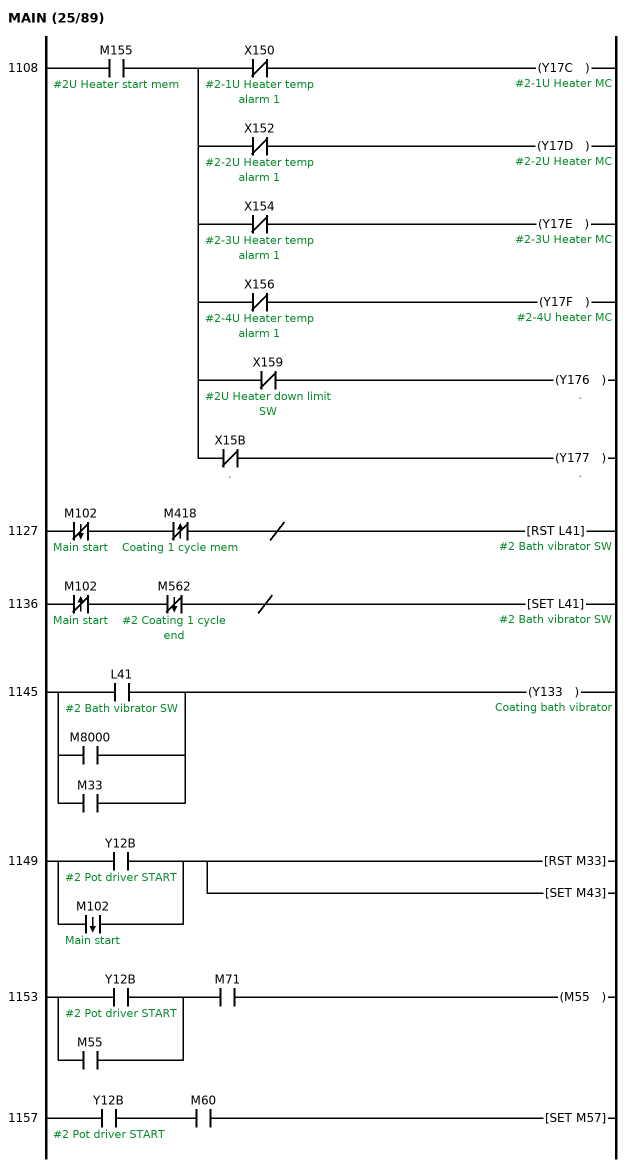
[picture p24: ladder of MAIN, rungs at steps 1108 to 1157]
1108  LD      M155  ; #2U Heater start mem
      MPS
      ANI     X150  ; #2-1U Heater temp alarm 1
      OUT     Y17C  ; #2-1U Heater MC
      MRD
      ANI     X152  ; #2-2U Heater temp alarm 1
      OUT     Y17D  ; #2-2U Heater MC
      MRD
      ANI     X154  ; #2-3U Heater temp alarm 1
      OUT     Y17E  ; #2-3U Heater MC
      MRD
      ANI     X156  ; #2-4U Heater temp alarm 1
      OUT     Y17F  ; #2-4U heater MC
      MRD
      ANI     X159  ; #2U Heater down limit SW
      OUT     Y176  ; .
      MPP
      ANI     X15B  ; .
      OUT     Y177  ; .
1127  LDFI    M102  ; Main start
      ANDPI   M418  ; Coating 1 cycle mem
      INV
      RST     L41  ; #2 Bath vibrator SW
1136  LDPI    M102  ; Main start
      ANDFI   M562  ; #2 Coating 1 cycle end
      INV
      SET     L41  ; #2 Bath vibrator SW
1145  LD      L41  ; #2 Bath vibrator SW
      OR      M8000
      OR      M33
      OUT     Y133  ; Coating bath vibrator
1149  LD      Y12B  ; #2 Pot driver START
      ORF     M102  ; Main start
      RST     M33
      SET     M43
1153  LD      Y12B  ; #2 Pot driver START
      OR      M55
      AND     M71
      OUT     M55
1157  LD      Y12B  ; #2 Pot driver START
      AND     M60
      SET     M57
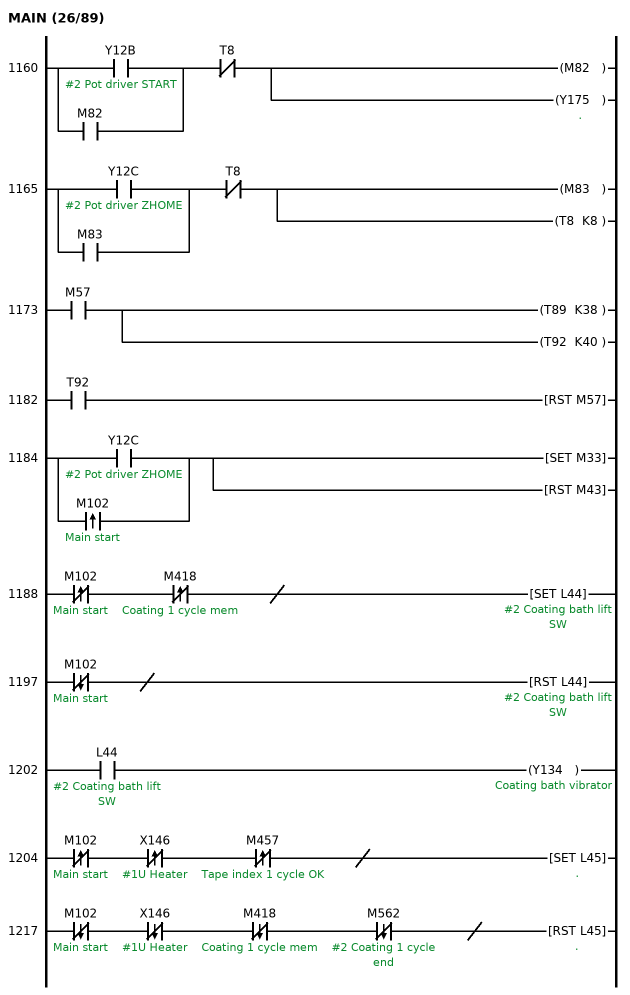
1160  LD      Y12B  ; #2 Pot driver START
      OR      M82
      ANI     T8
      OUT     M82
      OUT     Y175  ; .
1165  LD      Y12C  ; #2 Pot driver ZHOME
      OR      M83
      ANI     T8
      OUT     M83
      OUT     T8 K8
1173  LD      M57
      OUT     T89 K38
      OUT     T92 K40
1182  LD      T92
      RST     M57
1184  LD      Y12C  ; #2 Pot driver ZHOME
      ORP     M102  ; Main start
      SET     M33
      RST     M43
1188  LDPI    M102  ; Main start
      ANDPI   M418  ; Coating 1 cycle mem
      INV
      SET     L44  ; #2 Coating bath lift SW
1197  LDFI    M102  ; Main start
      INV
      RST     L44  ; #2 Coating bath lift SW
1202  LD      L44  ; #2 Coating bath lift SW
      OUT     Y134  ; Coating bath vibrator
1204  LDPI    M102  ; Main start
      ANDPI   X146  ; #1U Heater
      ANDPI   M457  ; Tape index 1 cycle OK
      INV
      SET     L45  ; .
1217  LDFI    M102  ; Main start
      ANDFI   X146  ; #1U Heater
      ANDFI   M418  ; Coating 1 cycle mem
      ANDFI   M562  ; #2 Coating 1 cycle end
      INV
      RST     L45  ; .
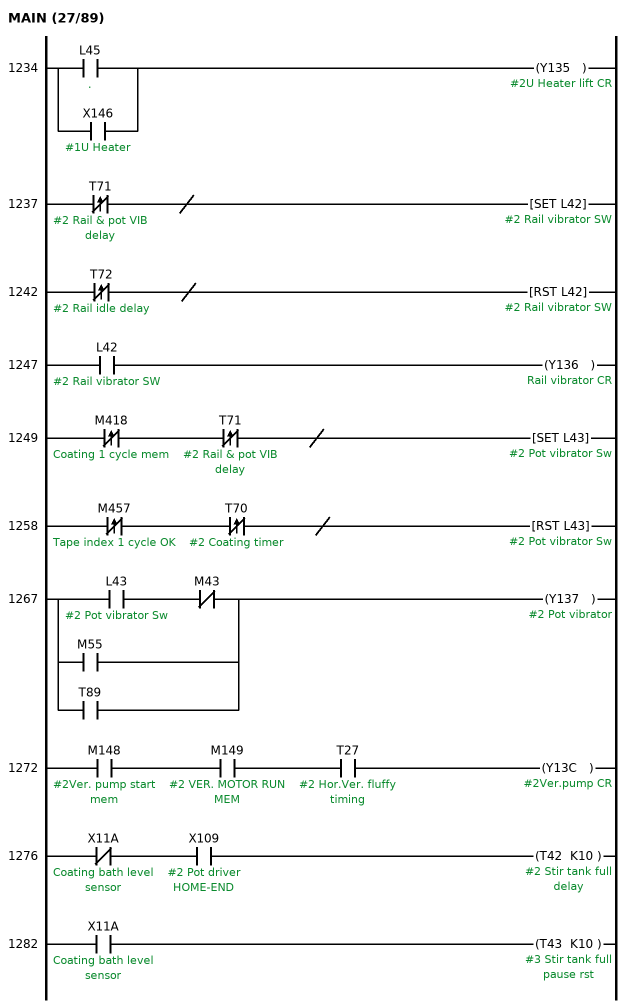
1234  LD      L45  ; .
      OR      X146  ; #1U Heater
      OUT     Y135  ; #2U Heater lift CR
1237  LDPI    T71  ; #2 Rail & pot VIB delay
      INV
      SET     L42  ; #2 Rail vibrator SW
1242  LDPI    T72  ; #2 Rail idle delay
      INV
      RST     L42  ; #2 Rail vibrator SW
1247  LD      L42  ; #2 Rail vibrator SW
      OUT     Y136  ; Rail vibrator CR
1249  LDPI    M418  ; Coating 1 cycle mem
      ANDPI   T71  ; #2 Rail & pot VIB delay
      INV
      SET     L43  ; #2 Pot vibrator Sw
1258  LDPI    M457  ; Tape index 1 cycle OK
      ANDPI   T70  ; #2 Coating timer
      INV
      RST     L43  ; #2 Pot vibrator Sw
1267  LD      L43  ; #2 Pot vibrator Sw
      ANI     M43
      OR      M55
      OR      T89
      OUT     Y137  ; #2 Pot vibrator
1272  LD      M148  ; #2Ver. pump start mem
      AND     M149  ; #2 VER. MOTOR RUN MEM
      AND     T27  ; #2 Hor.Ver. fluffy timing
      OUT     Y13C  ; #2Ver.pump CR
1276  LDI     X11A  ; Coating bath level sensor
      AND     X109  ; #2 Pot driver HOME-END
      OUT     T42 K10  ; #2 Stir tank full delay
1282  LD      X11A  ; Coating bath level sensor
      OUT     T43 K10  ; #3 Stir tank full pause rst
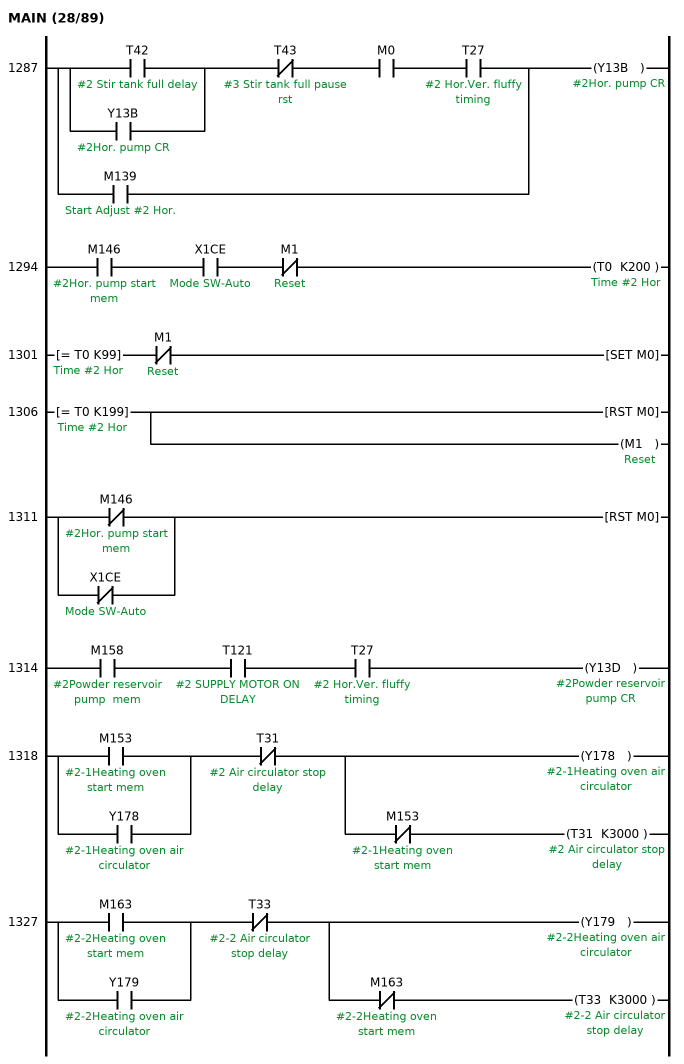
1287  LD      T42  ; #2 Stir tank full delay
      OR      Y13B  ; #2Hor. pump CR
      ANI     T43  ; #3 Stir tank full pause rst
      AND     M0
      AND     T27  ; #2 Hor.Ver. fluffy timing
      OR      M139  ; Start Adjust #2 Hor.
      OUT     Y13B  ; #2Hor. pump CR
1294  LD      M146  ; #2Hor. pump start mem
      AND     X1CE  ; Mode SW-Auto
      ANI     M1  ; Reset
      OUT     T0 K200  ; Time #2 Hor
1301  LD=     T0 K99  ; Time #2 Hor
      ANI     M1  ; Reset
      SET     M0
1306  LD=     T0 K199  ; Time #2 Hor
      RST     M0
      OUT     M1  ; Reset
1311  LDI     M146  ; #2Hor. pump start mem
      ORI     X1CE  ; Mode SW-Auto
      RST     M0
1314  LD      M158  ; #2Powder reservoir pump  mem
      AND     T121  ; #2 SUPPLY MOTOR ON DELAY
      AND     T27  ; #2 Hor.Ver. fluffy timing
      OUT     Y13D  ; #2Powder reservoir pump CR
1318  LD      M153  ; #2-1Heating oven start mem
      OR      Y178  ; #2-1Heating oven air circulator
      ANI     T31  ; #2 Air circulator stop delay
      OUT     Y178  ; #2-1Heating oven air circulator
      ANI     M153  ; #2-1Heating oven start mem
      OUT     T31 K3000  ; #2 Air circulator stop delay
1327  LD      M163  ; #2-2Heating oven start mem
      OR      Y179  ; #2-2Heating oven air circulator
      ANI     T33  ; #2-2 Air circulator stop delay
      OUT     Y179  ; #2-2Heating oven air circulator
      ANI     M163  ; #2-2Heating oven start mem
      OUT     T33 K3000  ; #2-2 Air circulator stop delay
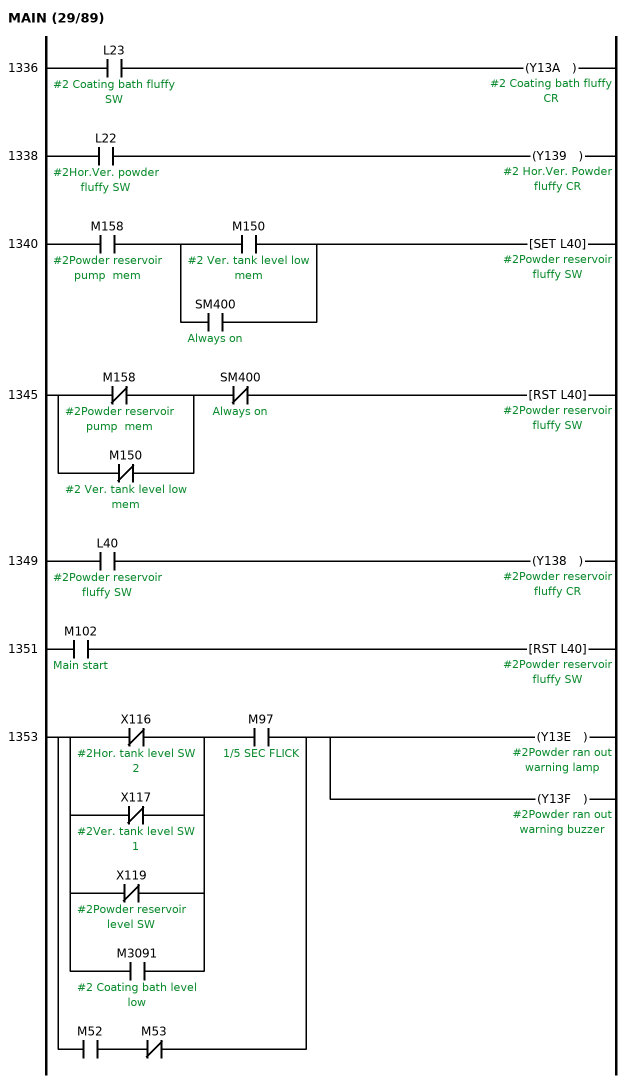
1336  LD      L23  ; #2 Coating bath fluffy SW
      OUT     Y13A  ; #2 Coating bath fluffy CR
1338  LD      L22  ; #2Hor.Ver. powder fluffy SW
      OUT     Y139  ; #2 Hor.Ver. Powder fluffy CR
1340  LD      M158  ; #2Powder reservoir pump  mem
      LD      M150  ; #2 Ver. tank level low mem
      OR      SM400  ; Always on
      ANB
      SET     L40  ; #2Powder reservoir fluffy SW
1345  LDI     M158  ; #2Powder reservoir pump  mem
      ORI     M150  ; #2 Ver. tank level low mem
      ANI     SM400  ; Always on
      RST     L40  ; #2Powder reservoir fluffy SW
1349  LD      L40  ; #2Powder reservoir fluffy SW
      OUT     Y138  ; #2Powder reservoir fluffy CR
1351  LD      M102  ; Main start
      RST     L40  ; #2Powder reservoir fluffy SW
1353  LDI     X116  ; #2Hor. tank level SW 2
      ORI     X117  ; #2Ver. tank level SW 1
      ORI     X119  ; #2Powder reservoir level SW
      OR      M3091  ; #2 Coating bath level low
      AND     M97  ; 1/5 SEC FLICK
      LD      M52
      ANI     M53
      ORB
      OUT     Y13E  ; #2Powder ran out warning lamp
      OUT     Y13F  ; #2Powder ran out warning buzzer
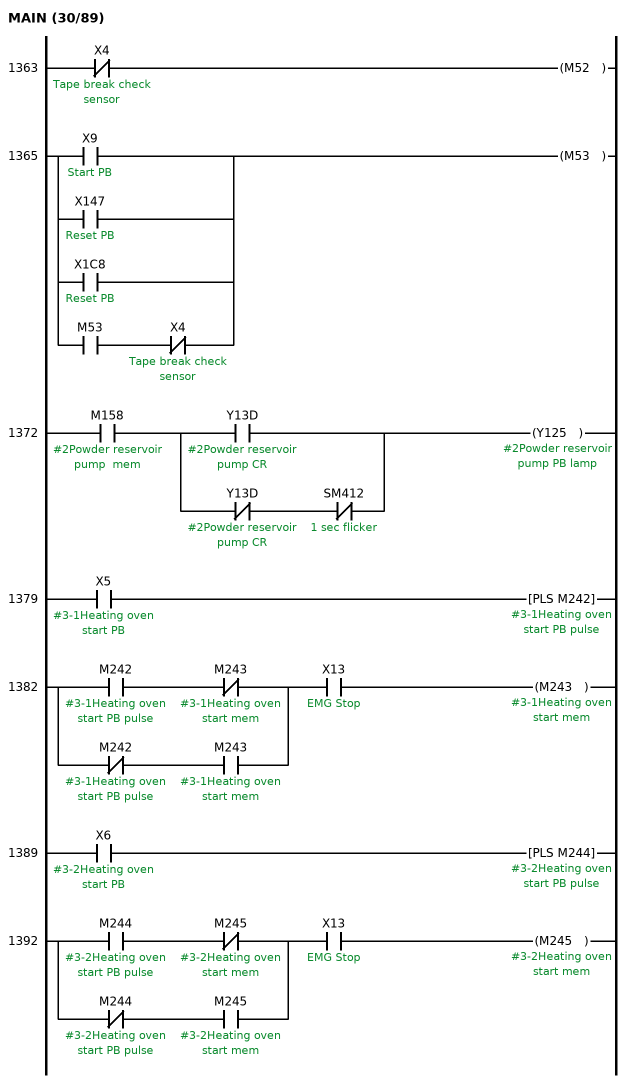
1363  LDI     X4  ; Tape break check sensor
      OUT     M52
1365  LD      X9  ; Start PB
      OR      X147  ; Reset PB
      OR      X1C8  ; Reset PB
      LD      M53
      ANI     X4  ; Tape break check sensor
      ORB
      OUT     M53
1372  LD      M158  ; #2Powder reservoir pump  mem
      LD      Y13D  ; #2Powder reservoir pump CR
      LDI     Y13D  ; #2Powder reservoir pump CR
      ANI     SM412  ; 1 sec flicker
      ORB
      ANB
      OUT     Y125  ; #2Powder reservoir pump PB lamp
1379  LD      X5  ; #3-1Heating oven start PB
      PLS     M242  ; #3-1Heating oven start PB pulse
1382  LD      M242  ; #3-1Heating oven start PB pulse
      ANI     M243  ; #3-1Heating oven start mem
      LDI     M242  ; #3-1Heating oven start PB pulse
      AND     M243  ; #3-1Heating oven start mem
      ORB
      AND     X13  ; EMG Stop
      OUT     M243  ; #3-1Heating oven start mem
1389  LD      X6  ; #3-2Heating oven start PB
      PLS     M244  ; #3-2Heating oven start PB pulse
1392  LD      M244  ; #3-2Heating oven start PB pulse
      ANI     M245  ; #3-2Heating oven start mem
      LDI     M244  ; #3-2Heating oven start PB pulse
      AND     M245  ; #3-2Heating oven start mem
      ORB
      AND     X13  ; EMG Stop
      OUT     M245  ; #3-2Heating oven start mem
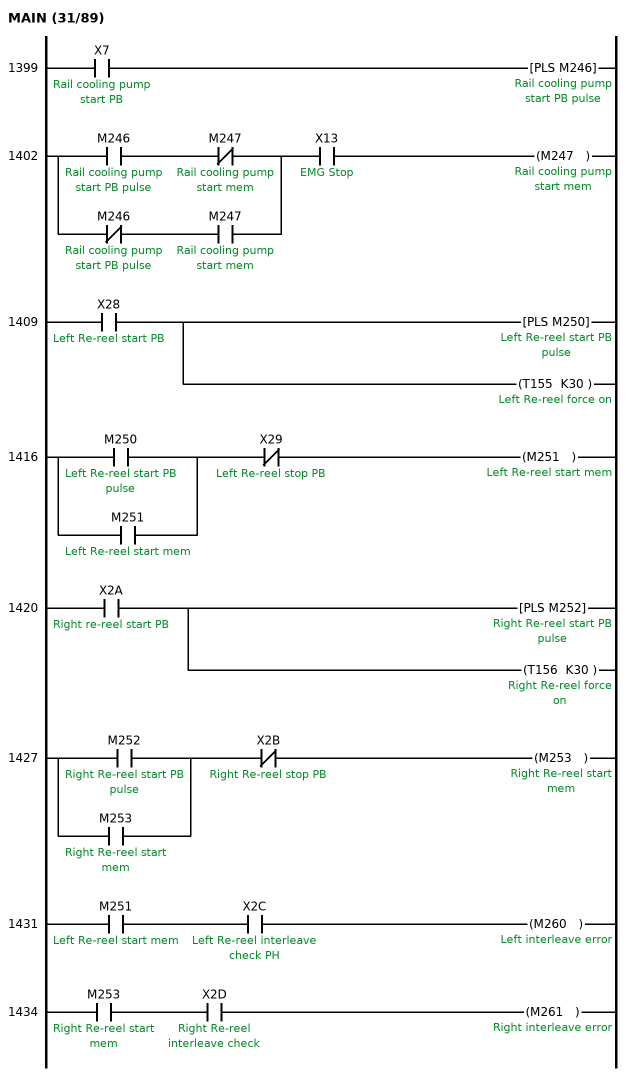
1399  LD      X7  ; Rail cooling pump start PB
      PLS     M246  ; Rail cooling pump start PB pulse
1402  LD      M246  ; Rail cooling pump start PB pulse
      ANI     M247  ; Rail cooling pump start mem
      LDI     M246  ; Rail cooling pump start PB pulse
      AND     M247  ; Rail cooling pump start mem
      ORB
      AND     X13  ; EMG Stop
      OUT     M247  ; Rail cooling pump start mem
1409  LD      X28  ; Left Re-reel start PB
      PLS     M250  ; Left Re-reel start PB pulse
      OUT     T155 K30  ; Left Re-reel force on
1416  LD      M250  ; Left Re-reel start PB pulse
      OR      M251  ; Left Re-reel start mem
      ANI     X29  ; Left Re-reel stop PB
      OUT     M251  ; Left Re-reel start mem
1420  LD      X2A  ; Right re-reel start PB
      PLS     M252  ; Right Re-reel start PB pulse
      OUT     T156 K30  ; Right Re-reel force on
1427  LD      M252  ; Right Re-reel start PB pulse
      OR      M253  ; Right Re-reel start mem
      ANI     X2B  ; Right Re-reel stop PB
      OUT     M253  ; Right Re-reel start mem
1431  LD      M251  ; Left Re-reel start mem
      AND     X2C  ; Left Re-reel interleave check PH
      OUT     M260  ; Left interleave error
1434  LD      M253  ; Right Re-reel start mem
      AND     X2D  ; Right Re-reel interleave check
      OUT     M261  ; Right interleave error
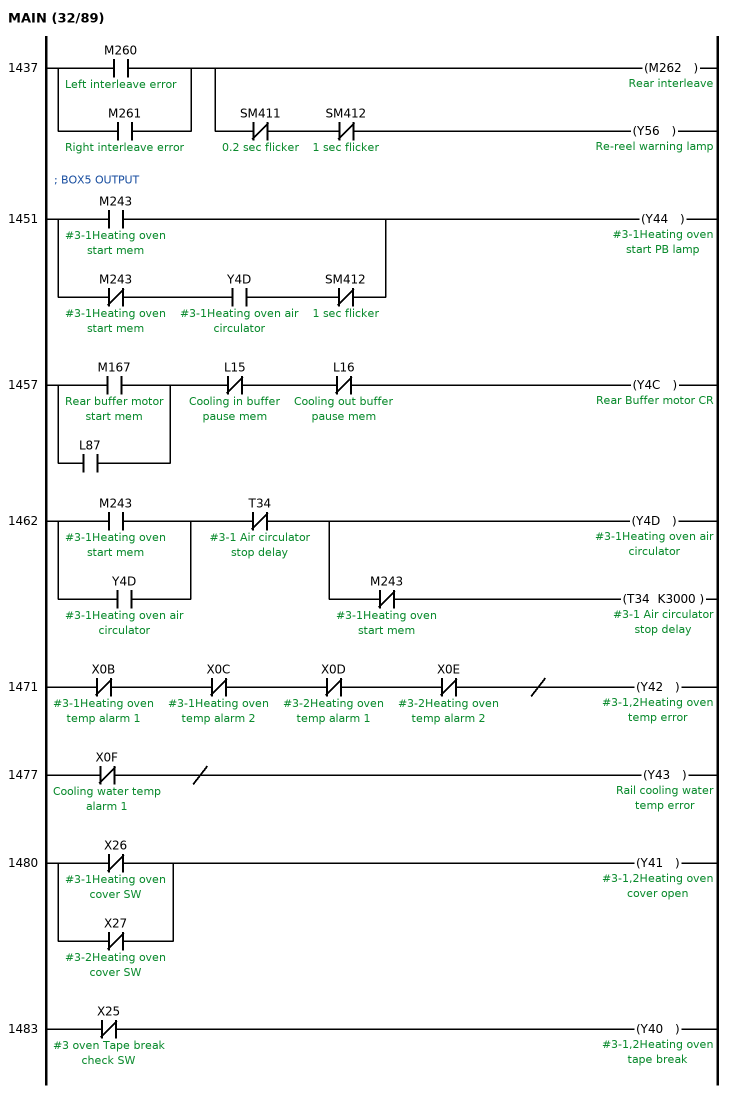
1437  LD      M260  ; Left interleave error
      OR      M261  ; Right interleave error
      OUT     M262  ; Rear interleave
      ANI     SM411  ; 0.2 sec flicker
      ANI     SM412  ; 1 sec flicker
      OUT     Y56  ; Re-reel warning lamp
; BOX5 OUTPUT
1451  LD      M243  ; #3-1Heating oven start mem
      LDI     M243  ; #3-1Heating oven start mem
      AND     Y4D  ; #3-1Heating oven air circulator
      ANI     SM412  ; 1 sec flicker
      ORB
      OUT     Y44  ; #3-1Heating oven start PB lamp
1457  LD      M167  ; Rear buffer motor start mem
      OR      L87
      ANI     L15  ; Cooling in buffer pause mem
      ANI     L16  ; Cooling out buffer pause mem
      OUT     Y4C  ; Rear Buffer motor CR
1462  LD      M243  ; #3-1Heating oven start mem
      OR      Y4D  ; #3-1Heating oven air circulator
      ANI     T34  ; #3-1 Air circulator stop delay
      OUT     Y4D  ; #3-1Heating oven air circulator
      ANI     M243  ; #3-1Heating oven start mem
      OUT     T34 K3000  ; #3-1 Air circulator stop delay
1471  LDI     X0B  ; #3-1Heating oven temp alarm 1
      ANI     X0C  ; #3-1Heating oven temp alarm 2
      ANI     X0D  ; #3-2Heating oven temp alarm 1
      ANI     X0E  ; #3-2Heating oven temp alarm 2
      INV
      OUT     Y42  ; #3-1,2Heating oven temp error
1477  LDI     X0F  ; Cooling water temp alarm 1
      INV
      OUT     Y43  ; Rail cooling water temp error
1480  LDI     X26  ; #3-1Heating oven cover SW
      ORI     X27  ; #3-2Heating oven cover SW
      OUT     Y41  ; #3-1,2Heating oven cover open
1483  LDI     X25  ; #3 oven Tape break check SW
      OUT     Y40  ; #3-1,2Heating oven tape break
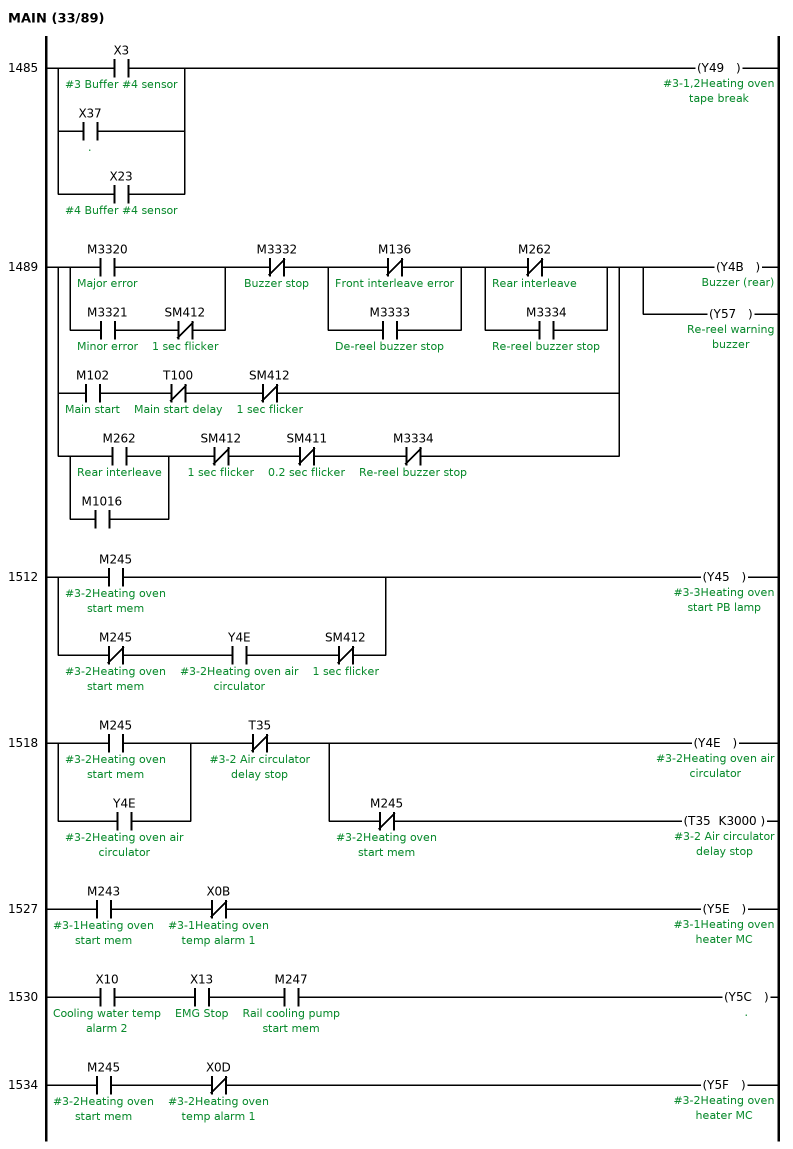
1485  LD      X3  ; #3 Buffer #4 sensor
      OR      X37  ; .
      OR      X23  ; #4 Buffer #4 sensor
      OUT     Y49  ; #3-1,2Heating oven tape break
1489  LD      M3320  ; Major error
      LD      M3321  ; Minor error
      ANI     SM412  ; 1 sec flicker
      ORB
      ANI     M3332  ; Buzzer stop
      LDI     M136  ; Front interleave error
      OR      M3333  ; De-reel buzzer stop
      ANB
      LDI     M262  ; Rear interleave
      OR      M3334  ; Re-reel buzzer stop
      ANB
      LD      M102  ; Main start
      ANI     T100  ; Main start delay
      ANI     SM412  ; 1 sec flicker
      ORB
      LD      M262  ; Rear interleave
      OR      M1016
      ANI     SM412  ; 1 sec flicker
      ANI     SM411  ; 0.2 sec flicker
      ANI     M3334  ; Re-reel buzzer stop
      ORB
      OUT     Y4B  ; Buzzer (rear)
      OUT     Y57  ; Re-reel warning buzzer
1512  LD      M245  ; #3-2Heating oven start mem
      LDI     M245  ; #3-2Heating oven start mem
      AND     Y4E  ; #3-2Heating oven air circulator
      ANI     SM412  ; 1 sec flicker
      ORB
      OUT     Y45  ; #3-3Heating oven start PB lamp
1518  LD      M245  ; #3-2Heating oven start mem
      OR      Y4E  ; #3-2Heating oven air circulator
      ANI     T35  ; #3-2 Air circulator delay stop
      OUT     Y4E  ; #3-2Heating oven air circulator
      ANI     M245  ; #3-2Heating oven start mem
      OUT     T35 K3000  ; #3-2 Air circulator delay stop
1527  LD      M243  ; #3-1Heating oven start mem
      ANI     X0B  ; #3-1Heating oven temp alarm 1
      OUT     Y5E  ; #3-1Heating oven heater MC
1530  LD      X10  ; Cooling water temp alarm 2
      AND     X13  ; EMG Stop
      AND     M247  ; Rail cooling pump start mem
      OUT     Y5C  ; .
1534  LD      M245  ; #3-2Heating oven start mem
      ANI     X0D  ; #3-2Heating oven temp alarm 1
      OUT     Y5F  ; #3-2Heating oven heater MC
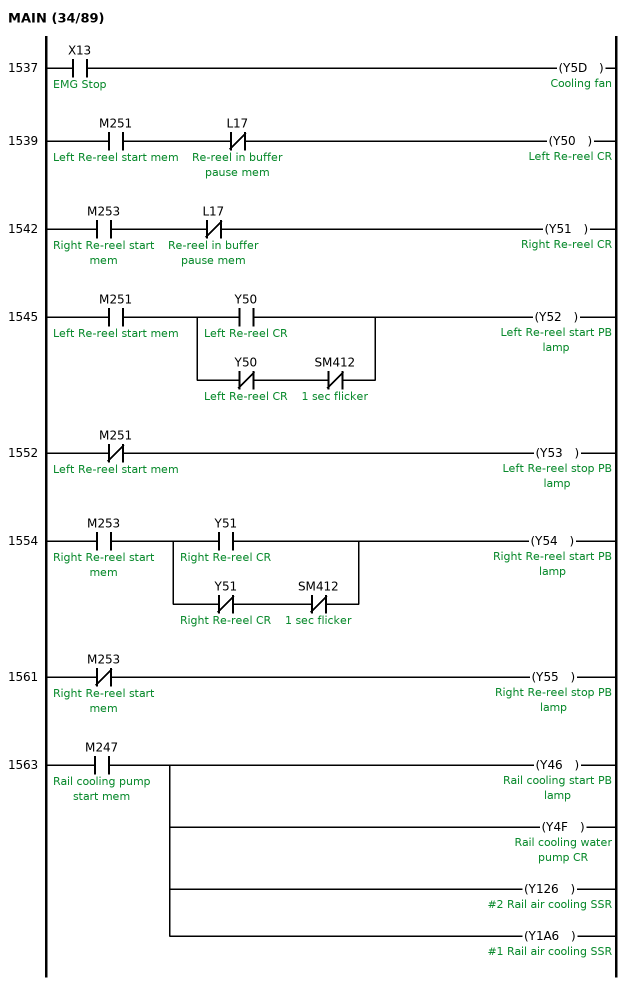
1537  LD      X13  ; EMG Stop
      OUT     Y5D  ; Cooling fan
1539  LD      M251  ; Left Re-reel start mem
      ANI     L17  ; Re-reel in buffer pause mem
      OUT     Y50  ; Left Re-reel CR
1542  LD      M253  ; Right Re-reel start mem
      ANI     L17  ; Re-reel in buffer pause mem
      OUT     Y51  ; Right Re-reel CR
1545  LD      M251  ; Left Re-reel start mem
      LD      Y50  ; Left Re-reel CR
      LDI     Y50  ; Left Re-reel CR
      ANI     SM412  ; 1 sec flicker
      ORB
      ANB
      OUT     Y52  ; Left Re-reel start PB lamp
1552  LDI     M251  ; Left Re-reel start mem
      OUT     Y53  ; Left Re-reel stop PB lamp
1554  LD      M253  ; Right Re-reel start mem
      LD      Y51  ; Right Re-reel CR
      LDI     Y51  ; Right Re-reel CR
      ANI     SM412  ; 1 sec flicker
      ORB
      ANB
      OUT     Y54  ; Right Re-reel start PB lamp
1561  LDI     M253  ; Right Re-reel start mem
      OUT     Y55  ; Right Re-reel stop PB lamp
1563  LD      M247  ; Rail cooling pump start mem
      OUT     Y46  ; Rail cooling start PB lamp
      OUT     Y4F  ; Rail cooling water pump CR
      OUT     Y126  ; #2 Rail air cooling SSR
      OUT     Y1A6  ; #1 Rail air cooling SSR
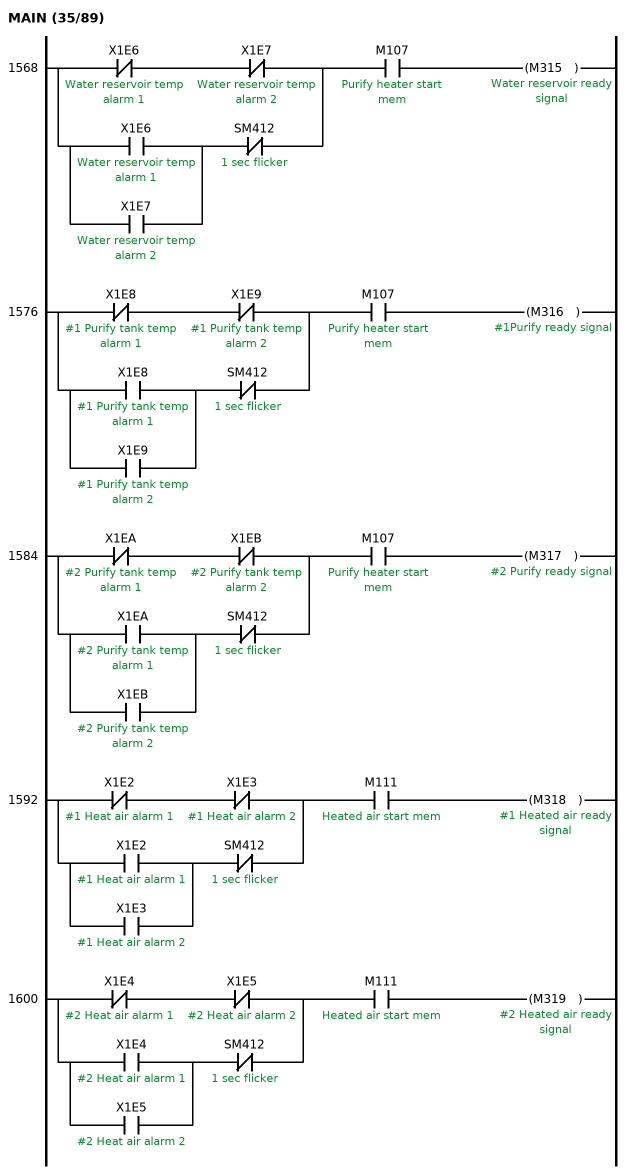
1568  LDI     X1E6  ; Water reservoir temp alarm 1
      ANI     X1E7  ; Water reservoir temp alarm 2
      LD      X1E6  ; Water reservoir temp alarm 1
      OR      X1E7  ; Water reservoir temp alarm 2
      ANI     SM412  ; 1 sec flicker
      ORB
      AND     M107  ; Purify heater start mem
      OUT     M315  ; Water reservoir ready signal
1576  LDI     X1E8  ; #1 Purify tank temp alarm 1
      ANI     X1E9  ; #1 Purify tank temp alarm 2
      LD      X1E8  ; #1 Purify tank temp alarm 1
      OR      X1E9  ; #1 Purify tank temp alarm 2
      ANI     SM412  ; 1 sec flicker
      ORB
      AND     M107  ; Purify heater start mem
      OUT     M316  ; #1Purify ready signal
1584  LDI     X1EA  ; #2 Purify tank temp alarm 1
      ANI     X1EB  ; #2 Purify tank temp alarm 2
      LD      X1EA  ; #2 Purify tank temp alarm 1
      OR      X1EB  ; #2 Purify tank temp alarm 2
      ANI     SM412  ; 1 sec flicker
      ORB
      AND     M107  ; Purify heater start mem
      OUT     M317  ; #2 Purify ready signal
1592  LDI     X1E2  ; #1 Heat air alarm 1
      ANI     X1E3  ; #1 Heat air alarm 2
      LD      X1E2  ; #1 Heat air alarm 1
      OR      X1E3  ; #1 Heat air alarm 2
      ANI     SM412  ; 1 sec flicker
      ORB
      AND     M111  ; Heated air start mem
      OUT     M318  ; #1 Heated air ready signal
1600  LDI     X1E4  ; #2 Heat air alarm 1
      ANI     X1E5  ; #2 Heat air alarm 2
      LD      X1E4  ; #2 Heat air alarm 1
      OR      X1E5  ; #2 Heat air alarm 2
      ANI     SM412  ; 1 sec flicker
      ORB
      AND     M111  ; Heated air start mem
      OUT     M319  ; #2 Heated air ready signal
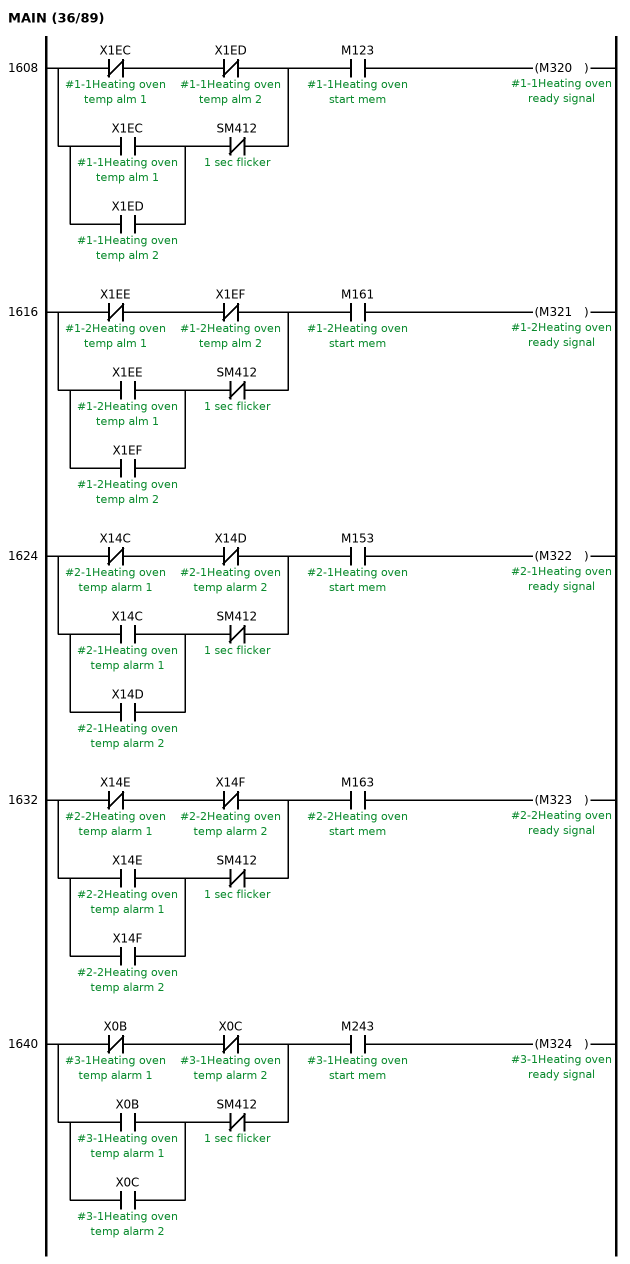
1608  LDI     X1EC  ; #1-1Heating oven temp alm 1
      ANI     X1ED  ; #1-1Heating oven temp alm 2
      LD      X1EC  ; #1-1Heating oven temp alm 1
      OR      X1ED  ; #1-1Heating oven temp alm 2
      ANI     SM412  ; 1 sec flicker
      ORB
      AND     M123  ; #1-1Heating oven start mem
      OUT     M320  ; #1-1Heating oven ready signal
1616  LDI     X1EE  ; #1-2Heating oven temp alm 1
      ANI     X1EF  ; #1-2Heating oven temp alm 2
      LD      X1EE  ; #1-2Heating oven temp alm 1
      OR      X1EF  ; #1-2Heating oven temp alm 2
      ANI     SM412  ; 1 sec flicker
      ORB
      AND     M161  ; #1-2Heating oven start mem
      OUT     M321  ; #1-2Heating oven ready signal
1624  LDI     X14C  ; #2-1Heating oven temp alarm 1
      ANI     X14D  ; #2-1Heating oven temp alarm 2
      LD      X14C  ; #2-1Heating oven temp alarm 1
      OR      X14D  ; #2-1Heating oven temp alarm 2
      ANI     SM412  ; 1 sec flicker
      ORB
      AND     M153  ; #2-1Heating oven start mem
      OUT     M322  ; #2-1Heating oven ready signal
1632  LDI     X14E  ; #2-2Heating oven temp alarm 1
      ANI     X14F  ; #2-2Heating oven temp alarm 2
      LD      X14E  ; #2-2Heating oven temp alarm 1
      OR      X14F  ; #2-2Heating oven temp alarm 2
      ANI     SM412  ; 1 sec flicker
      ORB
      AND     M163  ; #2-2Heating oven start mem
      OUT     M323  ; #2-2Heating oven ready signal
1640  LDI     X0B  ; #3-1Heating oven temp alarm 1
      ANI     X0C  ; #3-1Heating oven temp alarm 2
      LD      X0B  ; #3-1Heating oven temp alarm 1
      OR      X0C  ; #3-1Heating oven temp alarm 2
      ANI     SM412  ; 1 sec flicker
      ORB
      AND     M243  ; #3-1Heating oven start mem
      OUT     M324  ; #3-1Heating oven ready signal
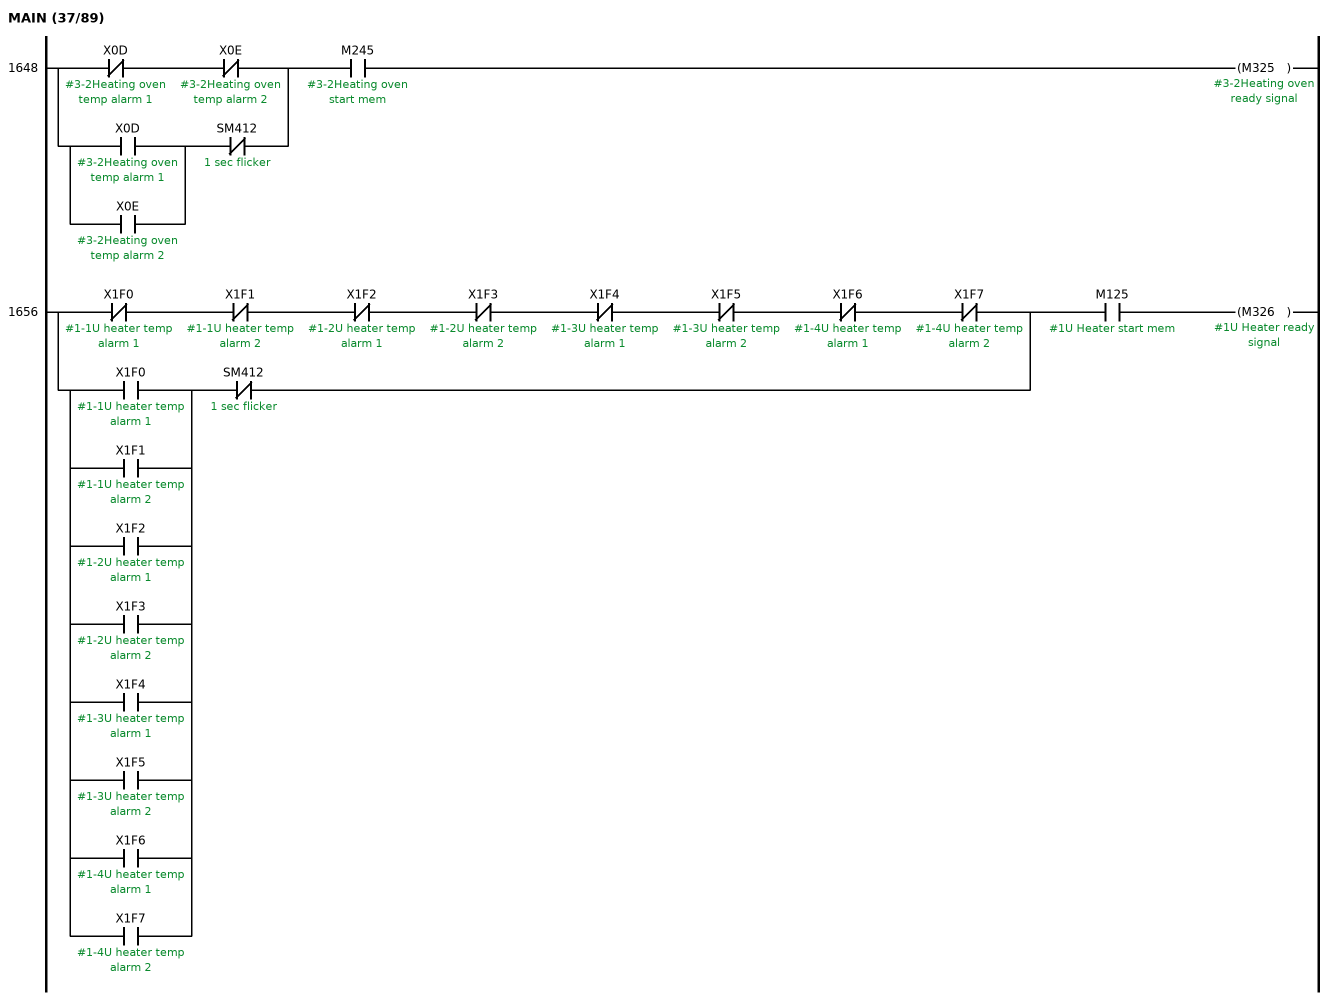
1648  LDI     X0D  ; #3-2Heating oven temp alarm 1
      ANI     X0E  ; #3-2Heating oven temp alarm 2
      LD      X0D  ; #3-2Heating oven temp alarm 1
      OR      X0E  ; #3-2Heating oven temp alarm 2
      ANI     SM412  ; 1 sec flicker
      ORB
      AND     M245  ; #3-2Heating oven start mem
      OUT     M325  ; #3-2Heating oven ready signal
1656  LDI     X1F0  ; #1-1U heater temp alarm 1
      ANI     X1F1  ; #1-1U heater temp alarm 2
      ANI     X1F2  ; #1-2U heater temp alarm 1
      ANI     X1F3  ; #1-2U heater temp alarm 2
      ANI     X1F4  ; #1-3U heater temp alarm 1
      ANI     X1F5  ; #1-3U heater temp alarm 2
      ANI     X1F6  ; #1-4U heater temp alarm 1
      ANI     X1F7  ; #1-4U heater temp alarm 2
      LD      X1F0  ; #1-1U heater temp alarm 1
      OR      X1F1  ; #1-1U heater temp alarm 2
      OR      X1F2  ; #1-2U heater temp alarm 1
      OR      X1F3  ; #1-2U heater temp alarm 2
      OR      X1F4  ; #1-3U heater temp alarm 1
      OR      X1F5  ; #1-3U heater temp alarm 2
      OR      X1F6  ; #1-4U heater temp alarm 1
      OR      X1F7  ; #1-4U heater temp alarm 2
      ANI     SM412  ; 1 sec flicker
      ORB
      AND     M125  ; #1U Heater start mem
      OUT     M326  ; #1U Heater ready signal
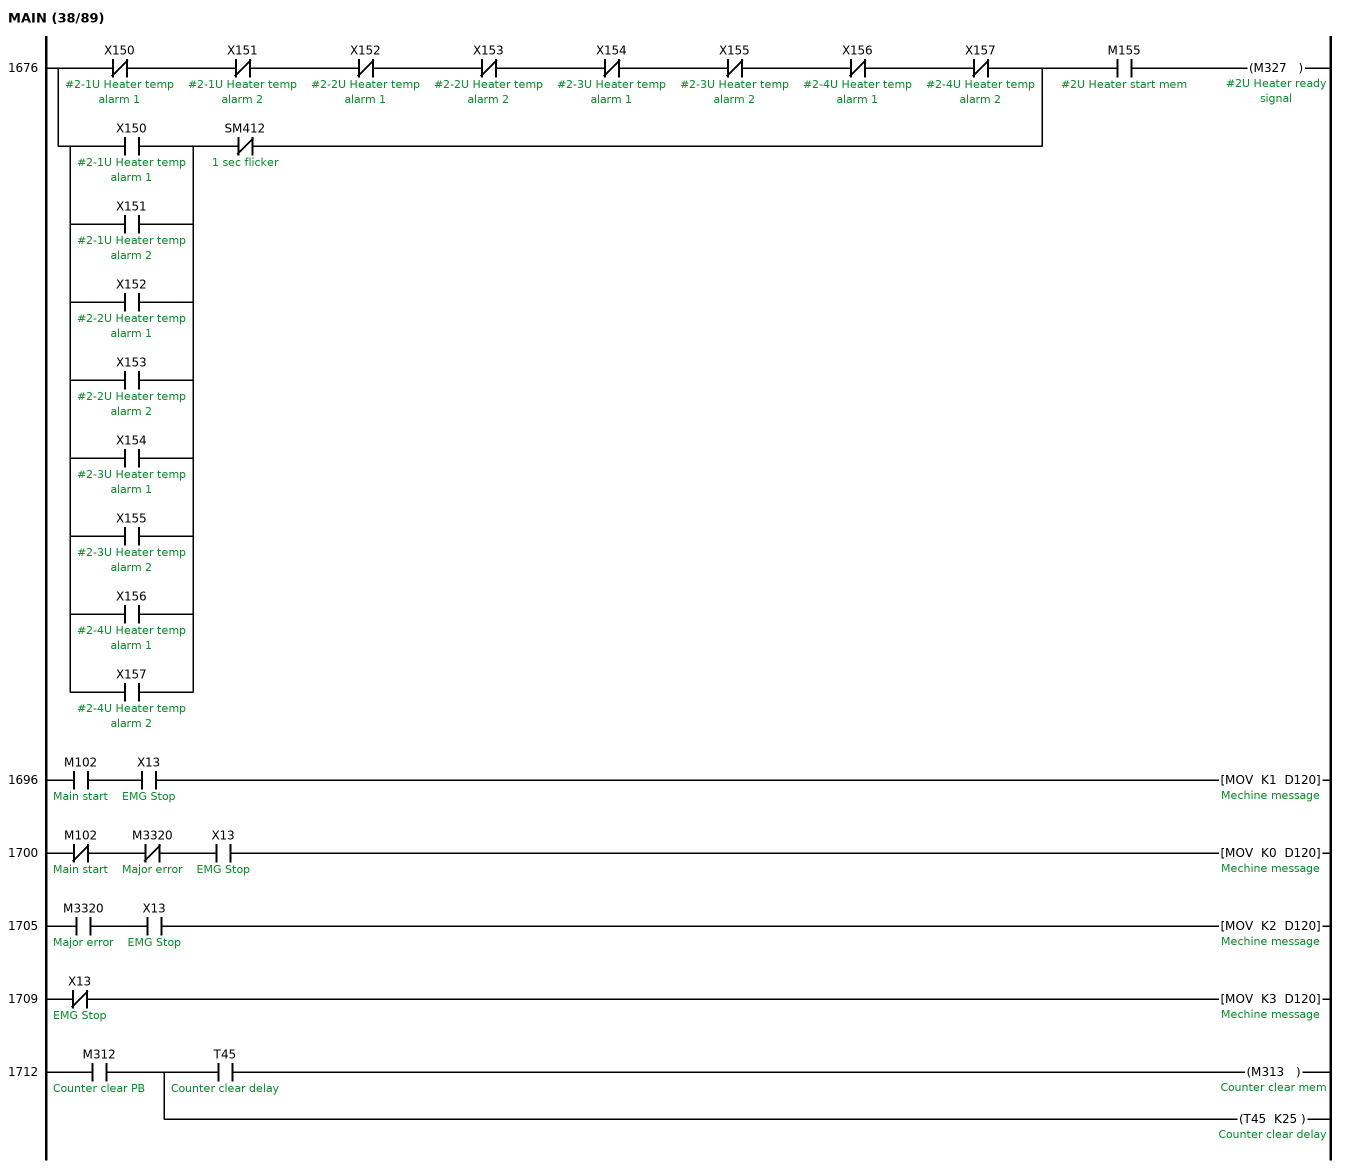
1676  LDI     X150  ; #2-1U Heater temp alarm 1
      ANI     X151  ; #2-1U Heater temp alarm 2
      ANI     X152  ; #2-2U Heater temp alarm 1
      ANI     X153  ; #2-2U Heater temp alarm 2
      ANI     X154  ; #2-3U Heater temp alarm 1
      ANI     X155  ; #2-3U Heater temp alarm 2
      ANI     X156  ; #2-4U Heater temp alarm 1
      ANI     X157  ; #2-4U Heater temp alarm 2
      LD      X150  ; #2-1U Heater temp alarm 1
      OR      X151  ; #2-1U Heater temp alarm 2
      OR      X152  ; #2-2U Heater temp alarm 1
      OR      X153  ; #2-2U Heater temp alarm 2
      OR      X154  ; #2-3U Heater temp alarm 1
      OR      X155  ; #2-3U Heater temp alarm 2
      OR      X156  ; #2-4U Heater temp alarm 1
      OR      X157  ; #2-4U Heater temp alarm 2
      ANI     SM412  ; 1 sec flicker
      ORB
      AND     M155  ; #2U Heater start mem
      OUT     M327  ; #2U Heater ready signal
1696  LD      M102  ; Main start
      AND     X13  ; EMG Stop
      MOV     K1 D120  ; Mechine message
1700  LDI     M102  ; Main start
      ANI     M3320  ; Major error
      AND     X13  ; EMG Stop
      MOV     K0 D120
1705  LD      M3320  ; Major error
      AND     X13  ; EMG Stop
      MOV     K2 D120
1709  LDI     X13  ; EMG Stop
      MOV     K3 D120
1712  LD      M312  ; Counter clear PB
      MPS
      AND     T45  ; Counter clear delay
      OUT     M313  ; Counter clear mem
      MPP
      OUT     T45 K25  ; Counter clear delay
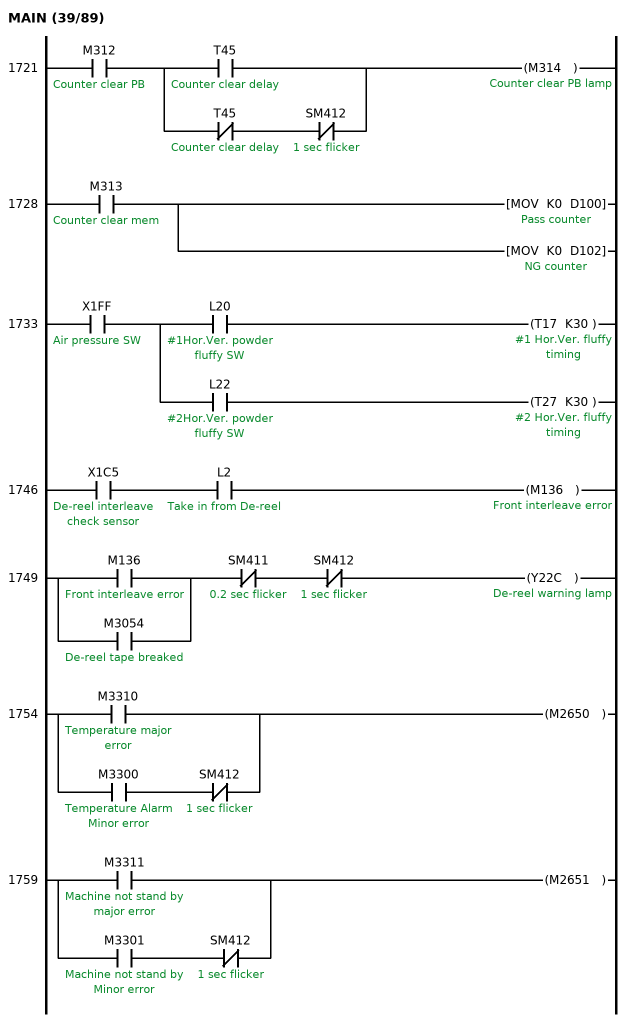
1721  LD      M312  ; Counter clear PB
      LD      T45  ; Counter clear delay
      LDI     T45  ; Counter clear delay
      ANI     SM412  ; 1 sec flicker
      ORB
      ANB
      OUT     M314  ; Counter clear PB lamp
1728  LD      M313  ; Counter clear mem
      MOV     K0 D100  ; Pass counter
      MOV     K0 D102  ; NG counter
1733  LD      X1FF  ; Air pressure SW
      MPS
      AND     L20  ; #1Hor.Ver. powder fluffy SW
      OUT     T17 K30  ; #1 Hor.Ver. fluffy timing
      MPP
      AND     L22  ; #2Hor.Ver. powder fluffy SW
      OUT     T27 K30  ; #2 Hor.Ver. fluffy timing
1746  LD      X1C5  ; De-reel interleave check sensor
      AND     L2  ; Take in from De-reel
      OUT     M136  ; Front interleave error
1749  LD      M136  ; Front interleave error
      OR      M3054  ; De-reel tape breaked
      ANI     SM411  ; 0.2 sec flicker
      ANI     SM412  ; 1 sec flicker
      OUT     Y22C  ; De-reel warning lamp
1754  LD      M3310  ; Temperature major error
      LD      M3300  ; Temperature Alarm Minor error
      ANI     SM412  ; 1 sec flicker
      ORB
      OUT     M2650
1759  LD      M3311  ; Machine not stand by major error
      LD      M3301  ; Machine not stand by Minor error
      ANI     SM412  ; 1 sec flicker
      ORB
      OUT     M2651
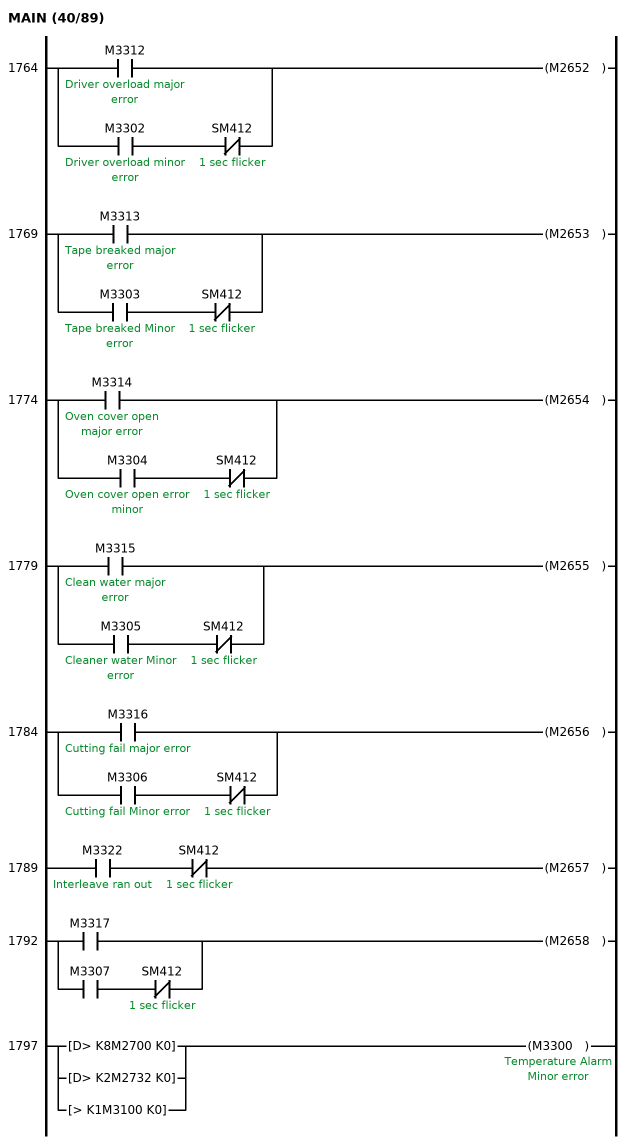
1764  LD      M3312  ; Driver overload major error
      LD      M3302  ; Driver overload minor error
      ANI     SM412  ; 1 sec flicker
      ORB
      OUT     M2652
1769  LD      M3313  ; Tape breaked major error
      LD      M3303  ; Tape breaked Minor error
      ANI     SM412  ; 1 sec flicker
      ORB
      OUT     M2653
1774  LD      M3314  ; Oven cover open major error
      LD      M3304  ; Oven cover open error minor
      ANI     SM412  ; 1 sec flicker
      ORB
      OUT     M2654
1779  LD      M3315  ; Clean water major error
      LD      M3305  ; Cleaner water Minor error
      ANI     SM412  ; 1 sec flicker
      ORB
      OUT     M2655
1784  LD      M3316  ; Cutting fail major error
      LD      M3306  ; Cutting fail Minor error
      ANI     SM412  ; 1 sec flicker
      ORB
      OUT     M2656
1789  LD      M3322  ; Interleave ran out
      ANI     SM412  ; 1 sec flicker
      OUT     M2657
1792  LD      M3317
      LD      M3307
      ANI     SM412  ; 1 sec flicker
      ORB
      OUT     M2658
1797  LDD>    K8M2700 K0  ; #1 Heated air alarm 1
      ORD>    K2M2732 K0  ; #2-2U heater high alarm
      OR>     K1M3100 K0  ; #1 Heated air alarm 1 Signal
      OUT     M3300  ; Temperature Alarm Minor error
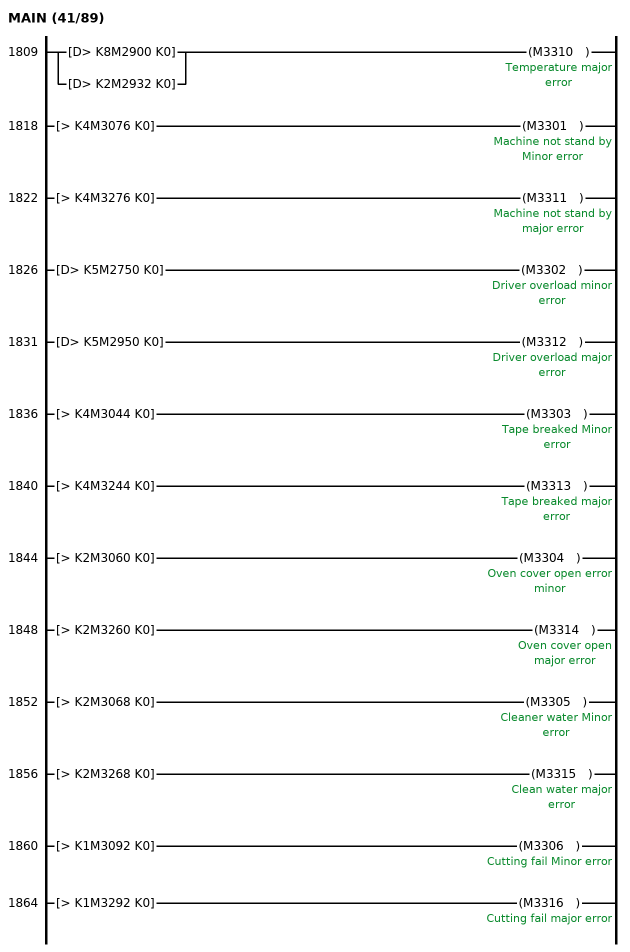
1809  LDD>    K8M2900 K0  ; #1 Heated air alarm 1
      ORD>    K2M2932 K0  ; #2-4U Heater temp alarm 1
      OUT     M3310  ; Temperature major error
1818  LD>     K4M3076 K0  ; Air low
      OUT     M3301  ; Machine not stand by Minor error
1822  LD>     K4M3276 K0  ; Air low mem
      OUT     M3311  ; Machine not stand by major error
1826  LDD>    K5M2750 K0  ; Heated air blower O.L
      OUT     M3302  ; Driver overload minor error
1831  LDD>    K5M2950 K0  ; Heated air driver O.L
      OUT     M3312  ; Driver overload major error
1836  LD>     K4M3044 K0  ; Front buffer tape breaked
      OUT     M3303  ; Tape breaked Minor error
1840  LD>     K4M3244 K0  ; Entry tape breaked mem
      OUT     M3313  ; Tape breaked major error
1844  LD>     K2M3060 K0  ; #1-1Heating  oven cover open
      OUT     M3304  ; Oven cover open error minor
1848  LD>     K2M3260 K0  ; #1-1Heating oven cover open mem
      OUT     M3314  ; Oven cover open major error
1852  LD>     K2M3068 K0  ; Water tank level low
      OUT     M3305  ; Cleaner water Minor error
1856  LD>     K2M3268 K0  ; Water tank level low mem
      OUT     M3315  ; Clean water major error
1860  LD>     K1M3092 K0  ; #1U Heater lift error
      OUT     M3306  ; Cutting fail Minor error
1864  LD>     K1M3292 K0  ; #1U Heater lift error
      OUT     M3316  ; Cutting fail major error
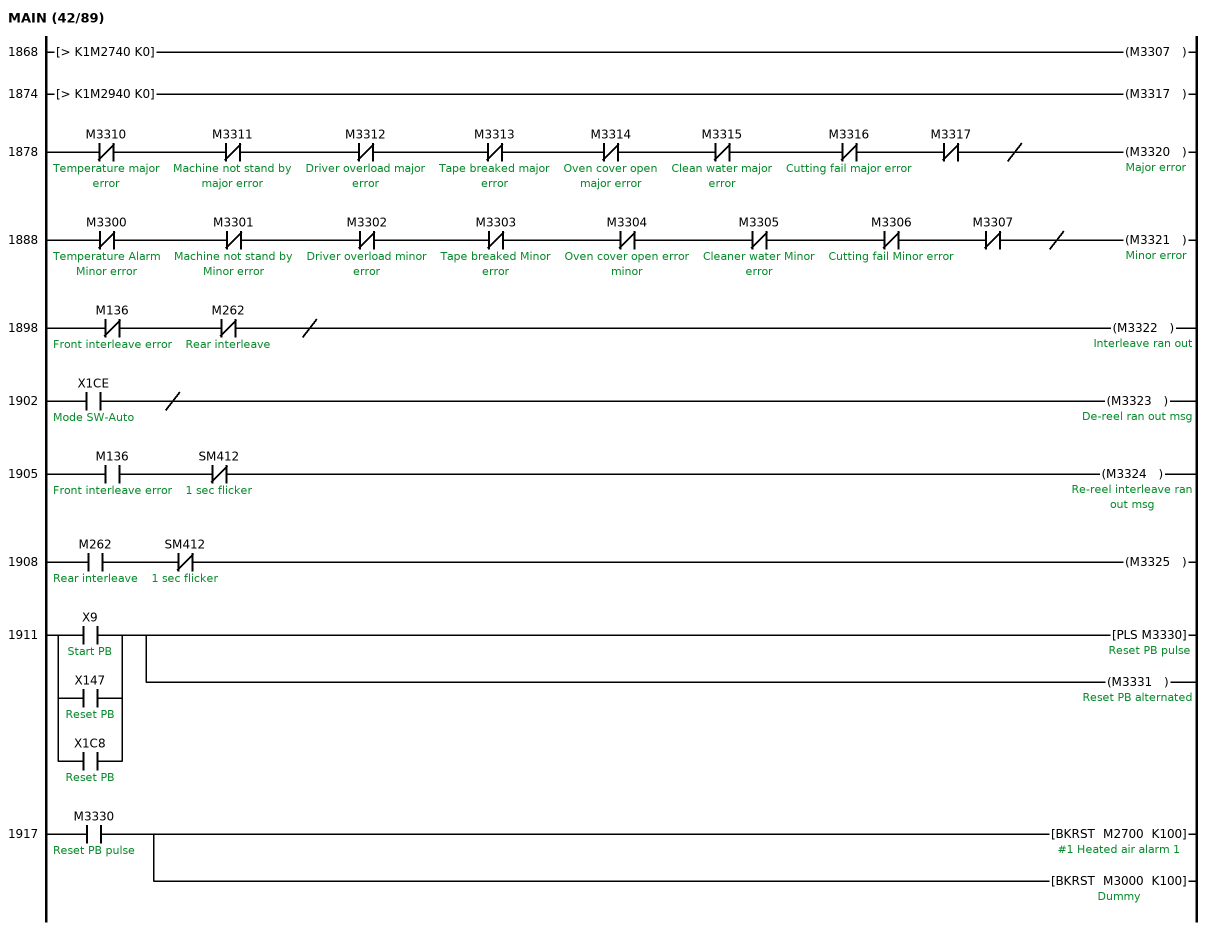
1868  LD>     K1M2740 K0
      OUT     M3307
        [note] 
1874  LD>     K1M2940 K0  ; .
      OUT     M3317
1878  LDI     M3310  ; Temperature major error
      ANI     M3311  ; Machine not stand by major error
      ANI     M3312  ; Driver overload major error
      ANI     M3313  ; Tape breaked major error
      ANI     M3314  ; Oven cover open major error
      ANI     M3315  ; Clean water major error
      ANI     M3316  ; Cutting fail major error
      ANI     M3317
      INV
      OUT     M3320  ; Major error
1888  LDI     M3300  ; Temperature Alarm Minor error
      ANI     M3301  ; Machine not stand by Minor error
      ANI     M3302  ; Driver overload minor error
      ANI     M3303  ; Tape breaked Minor error
      ANI     M3304  ; Oven cover open error minor
      ANI     M3305  ; Cleaner water Minor error
      ANI     M3306  ; Cutting fail Minor error
      ANI     M3307
      INV
      OUT     M3321  ; Minor error
1898  LDI     M136  ; Front interleave error
      ANI     M262  ; Rear interleave
      INV
      OUT     M3322  ; Interleave ran out
1902  LD      X1CE  ; Mode SW-Auto
      INV
      OUT     M3323  ; De-reel ran out msg
1905  LD      M136  ; Front interleave error
      ANI     SM412  ; 1 sec flicker
      OUT     M3324  ; Re-reel interleave ran out msg
1908  LD      M262  ; Rear interleave
      ANI     SM412  ; 1 sec flicker
      OUT     M3325
1911  LD      X9  ; Start PB
      OR      X147  ; Reset PB
      OR      X1C8  ; Reset PB
      PLS     M3330  ; Reset PB pulse
      OUT     M3331  ; Reset PB alternated
1917  LD      M3330  ; Reset PB pulse
      BKRST   M2700 K100
      BKRST   M3000 K100  ; Dummy
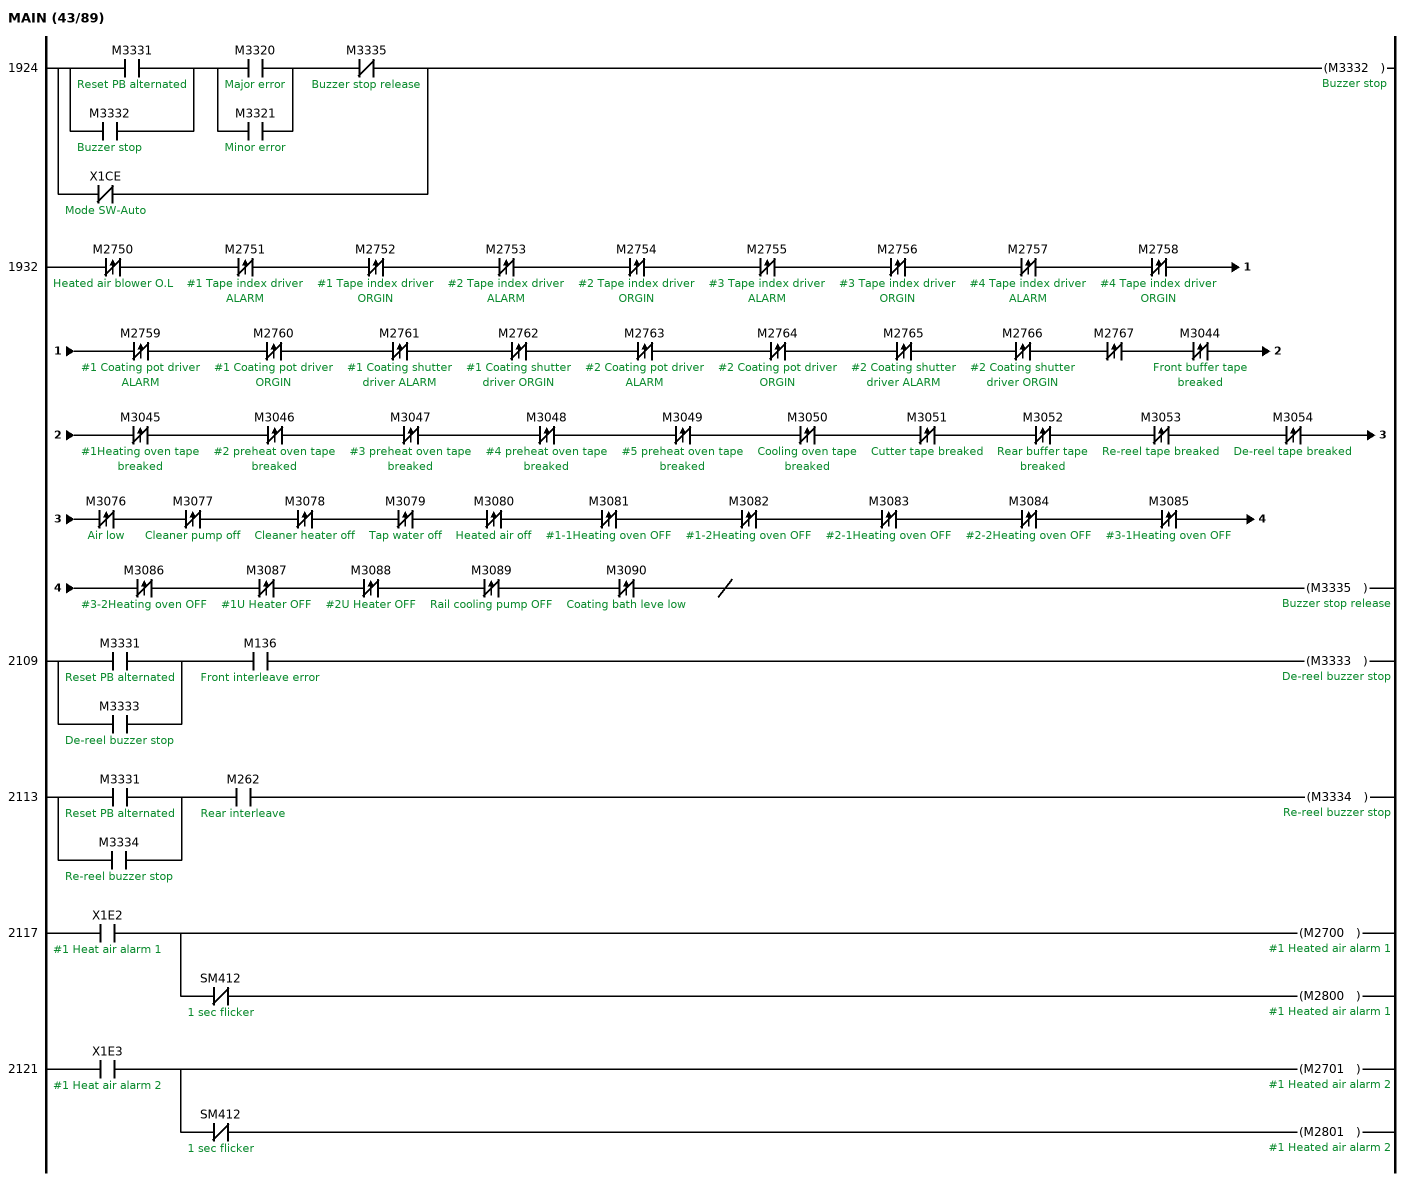
1924  LD      M3331  ; Reset PB alternated
      OR      M3332  ; Buzzer stop
      LD      M3320  ; Major error
      OR      M3321  ; Minor error
      ANB
      ANI     M3335  ; Buzzer stop release
      ORI     X1CE  ; Mode SW-Auto
      OUT     M3332  ; Buzzer stop
1932  LDPI    M2750  ; Heated air blower O.L
      ANDPI   M2751  ; #1 Tape index driver ALARM
      ANDPI   M2752  ; #1 Tape index driver ORGIN
      ANDPI   M2753  ; #2 Tape index driver ALARM
      ANDPI   M2754  ; #2 Tape index driver ORGIN
      ANDPI   M2755  ; #3 Tape index driver ALARM
      ANDPI   M2756  ; #3 Tape index driver ORGIN
      ANDPI   M2757  ; #4 Tape index driver ALARM
      ANDPI   M2758  ; #4 Tape index driver ORGIN
      ANDPI   M2759  ; #1 Coating pot driver ALARM
      ANDPI   M2760  ; #1 Coating pot driver ORGIN
      ANDPI   M2761  ; #1 Coating shutter driver ALARM
      ANDPI   M2762  ; #1 Coating shutter driver ORGIN
      ANDPI   M2763  ; #2 Coating pot driver ALARM
      ANDPI   M2764  ; #2 Coating pot driver ORGIN
      ANDPI   M2765  ; #2 Coating shutter driver ALARM
      ANDPI   M2766  ; #2 Coating shutter driver ORGIN
      ANDPI   M2767
      ANDPI   M3044  ; Front buffer tape breaked
      ANDPI   M3045  ; #1Heating oven tape breaked
      ANDPI   M3046  ; #2 preheat oven tape breaked
      ANDPI   M3047  ; #3 preheat oven tape breaked
      ANDPI   M3048  ; #4 preheat oven tape breaked
      ANDPI   M3049  ; #5 preheat oven tape breaked
      ANDPI   M3050  ; Cooling oven tape breaked
      ANDPI   M3051  ; Cutter tape breaked
      ANDPI   M3052  ; Rear buffer tape breaked
      ANDPI   M3053  ; Re-reel tape breaked
      ANDPI   M3054  ; De-reel tape breaked
      ANDPI   M3076  ; Air low
      ANDPI   M3077  ; Cleaner pump off
      ANDPI   M3078  ; Cleaner heater off
      ANDPI   M3079  ; Tap water off
      ANDPI   M3080  ; Heated air off
      ANDPI   M3081  ; #1-1Heating oven OFF
      ANDPI   M3082  ; #1-2Heating oven OFF
      ANDPI   M3083  ; #2-1Heating oven OFF
      ANDPI   M3084  ; #2-2Heating oven OFF
      ANDPI   M3085  ; #3-1Heating oven OFF
      ANDPI   M3086  ; #3-2Heating oven OFF
      ANDPI   M3087  ; #1U Heater OFF
      ANDPI   M3088  ; #2U Heater OFF
      ANDPI   M3089  ; Rail cooling pump OFF
      ANDPI   M3090  ; Coating bath leve low
      INV
      OUT     M3335  ; Buzzer stop release
2109  LD      M3331  ; Reset PB alternated
      OR      M3333  ; De-reel buzzer stop
      AND     M136  ; Front interleave error
      OUT     M3333  ; De-reel buzzer stop
2113  LD      M3331  ; Reset PB alternated
      OR      M3334  ; Re-reel buzzer stop
      AND     M262  ; Rear interleave
      OUT     M3334  ; Re-reel buzzer stop
2117  LD      X1E2  ; #1 Heat air alarm 1
      OUT     M2700  ; #1 Heated air alarm 1
      ANI     SM412  ; 1 sec flicker
      OUT     M2800  ; #1 Heated air alarm 1
2121  LD      X1E3  ; #1 Heat air alarm 2
      OUT     M2701  ; #1 Heated air alarm 2
      ANI     SM412  ; 1 sec flicker
      OUT     M2801  ; #1 Heated air alarm 2
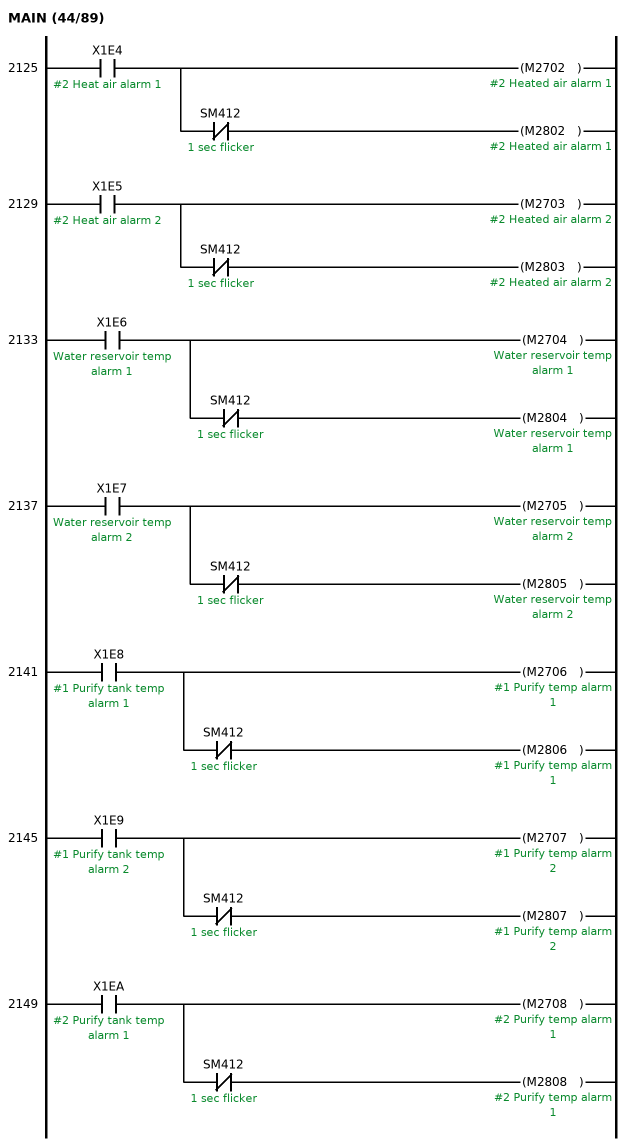
2125  LD      X1E4  ; #2 Heat air alarm 1
      OUT     M2702  ; #2 Heated air alarm 1
      ANI     SM412  ; 1 sec flicker
      OUT     M2802  ; #2 Heated air alarm 1
2129  LD      X1E5  ; #2 Heat air alarm 2
      OUT     M2703  ; #2 Heated air alarm 2
      ANI     SM412  ; 1 sec flicker
      OUT     M2803  ; #2 Heated air alarm 2
2133  LD      X1E6  ; Water reservoir temp alarm 1
      OUT     M2704  ; Water reservoir temp alarm 1
      ANI     SM412  ; 1 sec flicker
      OUT     M2804  ; Water reservoir temp alarm 1
2137  LD      X1E7  ; Water reservoir temp alarm 2
      OUT     M2705  ; Water reservoir temp alarm 2
      ANI     SM412  ; 1 sec flicker
      OUT     M2805  ; Water reservoir temp alarm 2
2141  LD      X1E8  ; #1 Purify tank temp alarm 1
      OUT     M2706  ; #1 Purify temp alarm 1
      ANI     SM412  ; 1 sec flicker
      OUT     M2806  ; #1 Purify temp alarm 1
2145  LD      X1E9  ; #1 Purify tank temp alarm 2
      OUT     M2707  ; #1 Purify temp alarm 2
      ANI     SM412  ; 1 sec flicker
      OUT     M2807  ; #1 Purify temp alarm 2
2149  LD      X1EA  ; #2 Purify tank temp alarm 1
      OUT     M2708  ; #2 Purify temp alarm 1
      ANI     SM412  ; 1 sec flicker
      OUT     M2808  ; #2 Purify temp alarm 1
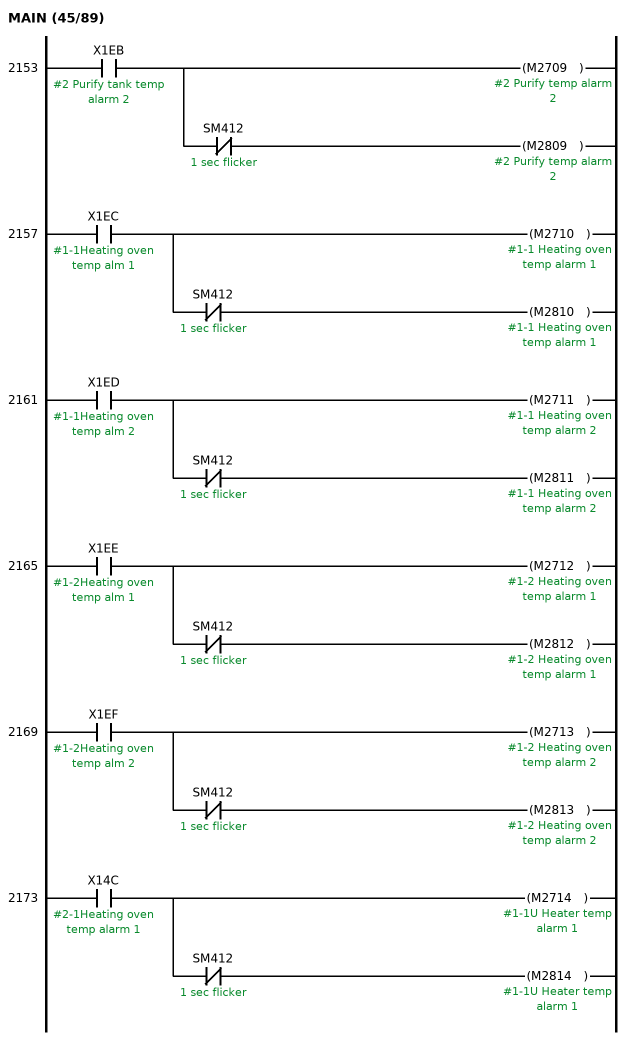
2153  LD      X1EB  ; #2 Purify tank temp alarm 2
      OUT     M2709  ; #2 Purify temp alarm 2
      ANI     SM412  ; 1 sec flicker
      OUT     M2809  ; #2 Purify temp alarm 2
2157  LD      X1EC  ; #1-1Heating oven temp alm 1
      OUT     M2710  ; #1-1 Heating oven temp alarm 1
      ANI     SM412  ; 1 sec flicker
      OUT     M2810  ; #1-1 Heating oven temp alarm 1
2161  LD      X1ED  ; #1-1Heating oven temp alm 2
      OUT     M2711  ; #1-1 Heating oven temp alarm 2
      ANI     SM412  ; 1 sec flicker
      OUT     M2811  ; #1-1 Heating oven temp alarm 2
2165  LD      X1EE  ; #1-2Heating oven temp alm 1
      OUT     M2712  ; #1-2 Heating oven temp alarm 1
      ANI     SM412  ; 1 sec flicker
      OUT     M2812  ; #1-2 Heating oven temp alarm 1
2169  LD      X1EF  ; #1-2Heating oven temp alm 2
      OUT     M2713  ; #1-2 Heating oven temp alarm 2
      ANI     SM412  ; 1 sec flicker
      OUT     M2813  ; #1-2 Heating oven temp alarm 2
2173  LD      X14C  ; #2-1Heating oven temp alarm 1
      OUT     M2714  ; #1-1U Heater temp alarm 1
      ANI     SM412  ; 1 sec flicker
      OUT     M2814  ; #1-1U Heater temp alarm 1
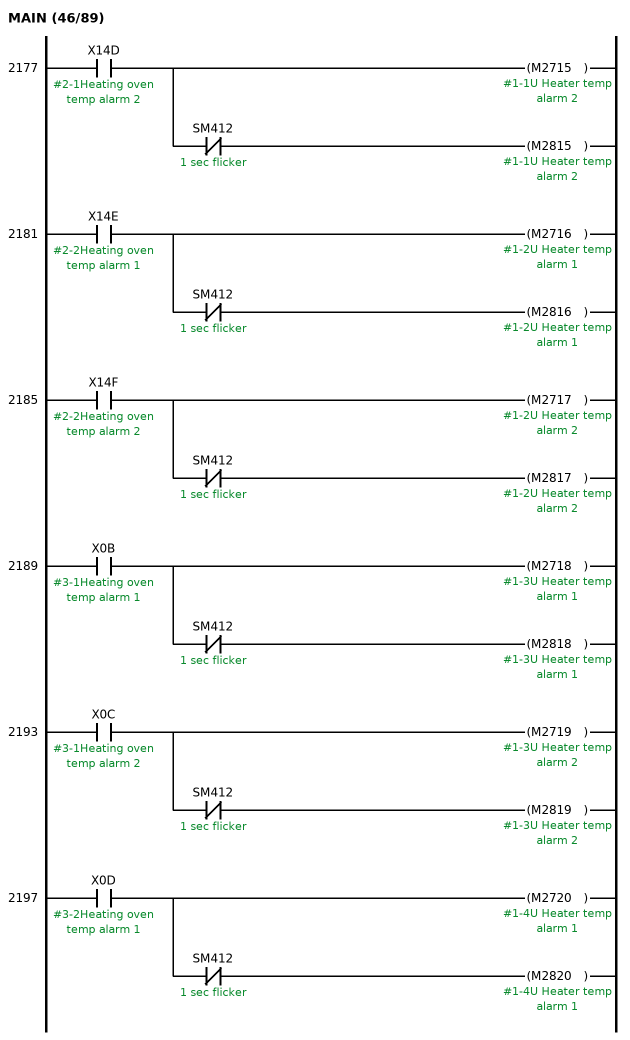
2177  LD      X14D  ; #2-1Heating oven temp alarm 2
      OUT     M2715  ; #1-1U Heater temp alarm 2
      ANI     SM412  ; 1 sec flicker
      OUT     M2815  ; #1-1U Heater temp alarm 2
2181  LD      X14E  ; #2-2Heating oven temp alarm 1
      OUT     M2716  ; #1-2U Heater temp alarm 1
      ANI     SM412  ; 1 sec flicker
      OUT     M2816  ; #1-2U Heater temp alarm 1
2185  LD      X14F  ; #2-2Heating oven temp alarm 2
      OUT     M2717  ; #1-2U Heater temp alarm 2
      ANI     SM412  ; 1 sec flicker
      OUT     M2817  ; #1-2U Heater temp alarm 2
2189  LD      X0B  ; #3-1Heating oven temp alarm 1
      OUT     M2718  ; #1-3U Heater temp alarm 1
      ANI     SM412  ; 1 sec flicker
      OUT     M2818  ; #1-3U Heater temp alarm 1
2193  LD      X0C  ; #3-1Heating oven temp alarm 2
      OUT     M2719  ; #1-3U Heater temp alarm 2
      ANI     SM412  ; 1 sec flicker
      OUT     M2819  ; #1-3U Heater temp alarm 2
2197  LD      X0D  ; #3-2Heating oven temp alarm 1
      OUT     M2720  ; #1-4U Heater temp alarm 1
      ANI     SM412  ; 1 sec flicker
      OUT     M2820  ; #1-4U Heater temp alarm 1
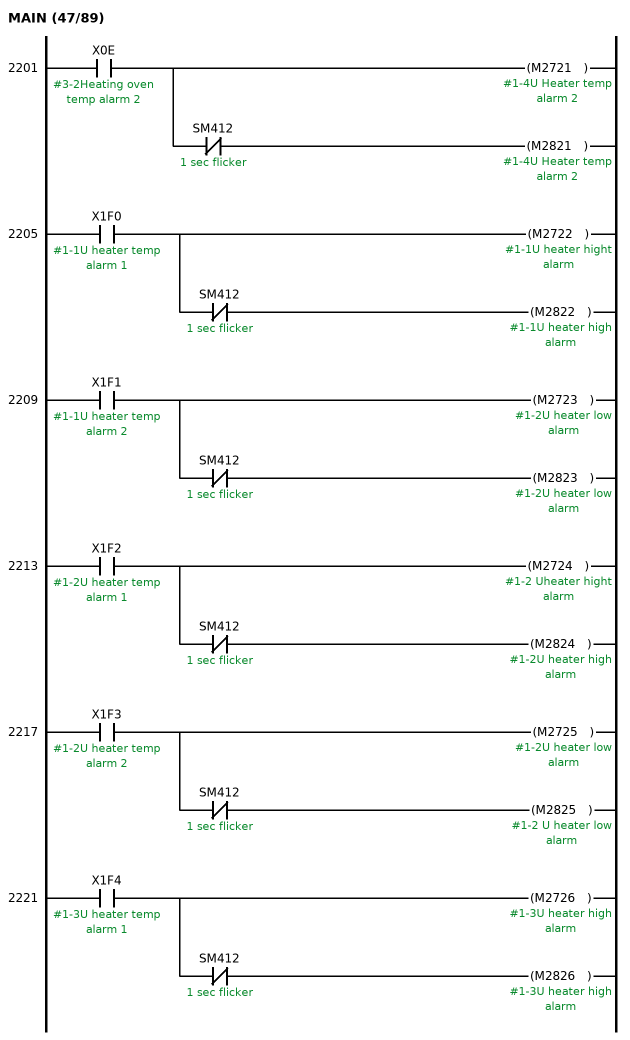
2201  LD      X0E  ; #3-2Heating oven temp alarm 2
      OUT     M2721  ; #1-4U Heater temp alarm 2
      ANI     SM412  ; 1 sec flicker
      OUT     M2821  ; #1-4U Heater temp alarm 2
2205  LD      X1F0  ; #1-1U heater temp alarm 1
      OUT     M2722  ; #1-1U heater hight alarm
      ANI     SM412  ; 1 sec flicker
      OUT     M2822  ; #1-1U heater high alarm
2209  LD      X1F1  ; #1-1U heater temp alarm 2
      OUT     M2723  ; #1-2U heater low alarm
      ANI     SM412  ; 1 sec flicker
      OUT     M2823  ; #1-2U heater low alarm
2213  LD      X1F2  ; #1-2U heater temp alarm 1
      OUT     M2724  ; #1-2 Uheater hight alarm
      ANI     SM412  ; 1 sec flicker
      OUT     M2824  ; #1-2U heater high alarm
2217  LD      X1F3  ; #1-2U heater temp alarm 2
      OUT     M2725  ; #1-2U heater low alarm
      ANI     SM412  ; 1 sec flicker
      OUT     M2825  ; #1-2 U heater low alarm
2221  LD      X1F4  ; #1-3U heater temp alarm 1
      OUT     M2726  ; #1-3U heater high alarm
      ANI     SM412  ; 1 sec flicker
      OUT     M2826  ; #1-3U heater high alarm
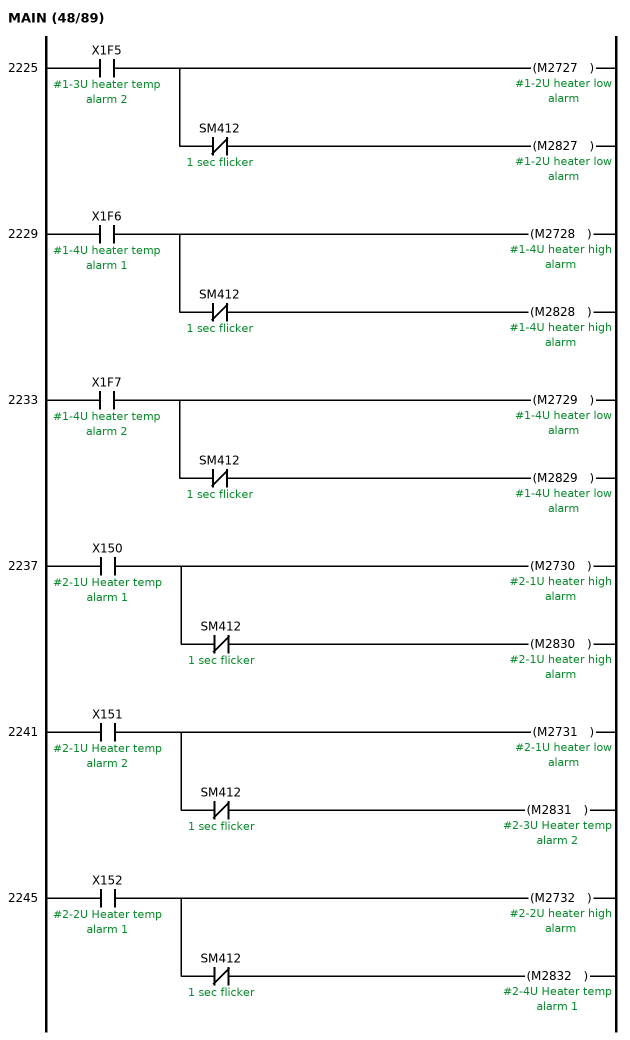
2225  LD      X1F5  ; #1-3U heater temp alarm 2
      OUT     M2727  ; #1-2U heater low alarm
      ANI     SM412  ; 1 sec flicker
      OUT     M2827  ; #1-2U heater low alarm
2229  LD      X1F6  ; #1-4U heater temp alarm 1
      OUT     M2728  ; #1-4U heater high alarm
      ANI     SM412  ; 1 sec flicker
      OUT     M2828  ; #1-4U heater high alarm
2233  LD      X1F7  ; #1-4U heater temp alarm 2
      OUT     M2729  ; #1-4U heater low alarm
      ANI     SM412  ; 1 sec flicker
      OUT     M2829  ; #1-4U heater low alarm
2237  LD      X150  ; #2-1U Heater temp alarm 1
      OUT     M2730  ; #2-1U heater high alarm
      ANI     SM412  ; 1 sec flicker
      OUT     M2830  ; #2-1U heater high alarm
2241  LD      X151  ; #2-1U Heater temp alarm 2
      OUT     M2731  ; #2-1U heater low alarm
      ANI     SM412  ; 1 sec flicker
      OUT     M2831  ; #2-3U Heater temp alarm 2
2245  LD      X152  ; #2-2U Heater temp alarm 1
      OUT     M2732  ; #2-2U heater high alarm
      ANI     SM412  ; 1 sec flicker
      OUT     M2832  ; #2-4U Heater temp alarm 1
